// TIA Portal V19 export
TYPE "udt_RollLubr_Valve_Pers"
   STRUCT
      SystemOn : Bool;
      Enable_V : Array[1.."ROLL_LUBR_MAXVALVE"] of Bool;
      TimeOn : Time;
      TimeOff : Time;
   END_STRUCT;
END_TYPE
